// TIA Portal project "Testing" (V15.1)

(* hardware
DEVICE "S71500/ET200MP station_1"  S7-1500 station
   slot 0: "Rail_0"  Rack  6ES7 590-1***0-0AA0
   slot 1: "PLC_1"  CPU 1513-1 PN  6ES7 513-1AL02-0AB0  V2.6
      slot 3: "CPU display_1"  6ES7591-1AA00-0AA0
*)

// ===== PLC "PLC_1"  CPU 1513-1 PN =====

DATA_BLOCK "Auxiliare"   // DB1
{ S7_Optimized_Access := 'TRUE' }
VERSION : 0.1
   VAR
      btn_trigger : Bool;
      aux_1 : Bool;
      aux_2 : Bool;
      counter_1 : DInt;
      counter_2 : DInt;
   END_VAR
BEGIN
END_DATA_BLOCK

ORGANIZATION_BLOCK "Main"   // OB1, LAD, ProgramCycle
TITLE = "Main Program Sweep (Cycle)"
{ S7_Optimized_Access := 'TRUE' }
VERSION : 0.1
   VAR_INPUT
      Initial_Call : Bool;   // Initial call of this OB
      Remanence : Bool;   // =True, if remanent data are available
   END_VAR
   VAR_TEMP   // added for the SCL form of the ladder/FBD networks
      _w1 : Bool;
   END_VAR
BEGIN

REGION Network 1: positive edge
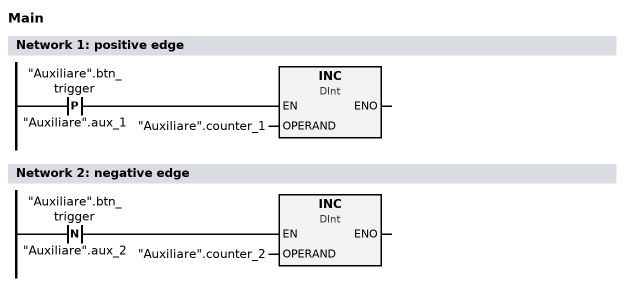
   RUNG wire#powerrail
      P_Contact(operand := "Auxiliare".btn_trigger, bit := "Auxiliare".aux_1)
      { S7_Templates := "DestType := DInt" } Inc( "Auxiliare".counter_1 )
   END_RUNG
   // the same network as SCL:
   #_w1 := "Auxiliare".btn_trigger AND NOT "Auxiliare".aux_1;   // rising edge of "Auxiliare".btn_trigger
   "Auxiliare".aux_1 := "Auxiliare".btn_trigger;
   IF #_w1 THEN "Auxiliare".counter_1 := "Auxiliare".counter_1 + 1; END_IF;
END_REGION

REGION Network 2: negative edge
   RUNG wire#powerrail
      N_Contact(operand := "Auxiliare".btn_trigger, bit := "Auxiliare".aux_2)
      { S7_Templates := "DestType := DInt" } Inc( "Auxiliare".counter_2 )
   END_RUNG
   // the same network as SCL:
   #_w1 := NOT "Auxiliare".btn_trigger AND "Auxiliare".aux_2;   // falling edge of "Auxiliare".btn_trigger
   "Auxiliare".aux_2 := "Auxiliare".btn_trigger;
   IF #_w1 THEN "Auxiliare".counter_2 := "Auxiliare".counter_2 + 1; END_IF;
END_REGION
END_ORGANIZATION_BLOCK